// TwinCAT 3 PLC project Command_Pattern
// ProgramVersion: 3.1.4024.0
// libraries:
//   Tc2_Standard, * (Beckhoff Automation GmbH)
//   Tc2_System, * (Beckhoff Automation GmbH)
//   Tc2_Utilities, * (Beckhoff Automation GmbH)
//   Tc3_Module, * (Beckhoff Automation GmbH)
// project tree:
//   Commands/ AxisDisableCommand.TcPOU, AxisEnableCommand.TcPOU, AxisMoveCommand.TcPOU, ITF_Command.TcIO
//   Invoker/ Invoker.TcPOU
//   / PlcTask.TcTTO
//   POUs/ MAIN.TcPOU
//   Reciever/ FB_Axis.TcPOU, ITF_Axis.TcIO
// (motion and I/O tree: see PLC project simple_factory_pattern)
// real-time tasks:
//   TASK PlcTask: cycle T#10ms, priority 20, ADS port 350
//   TASK PlcTask1: cycle T#10ms, priority 21, ADS port 351
//   TASK PlcTask2: cycle T#10ms, priority 22, ADS port 352
//   TASK PlcTask3: cycle T#10ms, priority 23, ADS port 353
//   TASK PlcTask4: cycle T#10ms, priority 24, ADS port 354
//   TASK PlcTask5: cycle T#10ms, priority 25, ADS port 355
//   TASK PlcTask6: cycle T#10ms, priority 26, ADS port 356
//   TASK PlcTask7: cycle T#10ms, priority 27, ADS port 357
//   TASK PlcTask8: cycle T#10ms, priority 28, ADS port 358
//   TASK PlcTask9: cycle T#10ms, priority 29, ADS port 359
//   TASK PlcTask10: cycle T#10ms, priority 30, ADS port 360
//   TASK PlcTask11: cycle T#10ms, priority 31, ADS port 361

CONFIGURATION Command_Pattern
    RESOURCE PLC ON TwinCAT3
        TASK PlcTask(INTERVAL := T#10ms, PRIORITY := 30);
        PROGRAM MAIN WITH PlcTask : MAIN;
    END_RESOURCE
END_CONFIGURATION

// ---- Commands/ITF_Command.TcIO
INTERFACE ITF_Command

METHOD Execute : BOOL
VAR_INPUT
END_VAR
END_METHOD

END_INTERFACE

// ---- Reciever/ITF_Axis.TcIO
INTERFACE ITF_Axis

METHOD Disable : BOOL
VAR_INPUT
END_VAR
END_METHOD

METHOD Enable : BOOL
VAR_INPUT
	EnablePositive : BOOL;
	EnableNegative : BOOL;
	Override : LREAL;
END_VAR
END_METHOD

METHOD MoveToPosition : BOOL
VAR_INPUT
	Position : LREAL;
	Velocity : LREAL;
END_VAR
END_METHOD

END_INTERFACE

// ---- POUs/MAIN.TcPOU
PROGRAM MAIN
VAR
	Axis1 : FB_Axis;
	DisableCmd : AxisDisableCommand := (MyAxis := Axis1);
	EnableCmd : AxisEnableCommand := (MyAxis := Axis1);
	MoveCmd : AxisMoveCommand := (MyAxis := Axis1);
	EnableButton : Invoker;
	DisableButton : Invoker;
	MoveButton : Invoker;
	Initialised: BOOL;
	Enable: BOOL;
	Disable: BOOL;
	MoveAxis: BOOL;
END_VAR

IF NOT Initialised THEN
	EnableButton.SetCommand(MyCommand := EnableCmd);
	DisableButton.SetCommand(MyCommand := DisableCmd);
	MoveButton.SetCommand(MyCommand := MoveCmd);
	Initialised := TRUE;
END_IF

IF Enable THEN
	IF EnableButton.ExecuteCommand() THEN
		Enable := FALSE;
	END_IF
END_IF

IF Disable THEN
	IF DisableButton.ExecuteCommand() THEN
		Disable := FALSE;
	END_IF
END_IF

IF MoveAxis THEN
	IF MoveButton.ExecuteCommand() THEN
		MoveAxis := FALSE;
	END_IF
END_IF

END_PROGRAM

// ---- Reciever/FB_Axis.TcPOU
FUNCTION_BLOCK PUBLIC FB_Axis IMPLEMENTS ITF_Axis
VAR
	testString : STRING;
END_VAR

METHOD Disable : BOOL
VAR_INPUT
END_VAR
ADSLOGSTR( msgCtrlMask := ADSLOG_MSGTYPE_ERROR OR ADSLOG_MSGTYPE_MSGBOX,
			msgFmtStr :='Axis Disabling',
 			strArg := '');
END_METHOD

METHOD Enable : BOOL
VAR_INPUT
	EnablePositive : BOOL;
	EnableNegative : BOOL;
	Override : LREAL;
END_VAR
testString := '';
testString := CONCAT(testString, '[');
testString := CONCAT(testString, BOOL_TO_STRING(EnablePositive));
testString := CONCAT(testString, ']');
testString := CONCAT(testString, '[');
testString := CONCAT(testString, BOOL_TO_STRING(EnableNegative));
testString := CONCAT(testString, ']');
testString := CONCAT(testString, '[');
testString := CONCAT(testString, LREAL_TO_STRING(Override));
testString := CONCAT(testString, ']');

ADSLOGSTR( msgCtrlMask := ADSLOG_MSGTYPE_ERROR OR ADSLOG_MSGTYPE_MSGBOX,
			msgFmtStr :='Axis Enabling: %s',
 			strArg := testString);
END_METHOD

METHOD MoveToPosition : BOOL
VAR_INPUT
	Position : LREAL;
	Velocity : LREAL;
END_VAR
testString := '';
testString := CONCAT(testString, '[');
testString := CONCAT(testString, LREAL_TO_STRING(Position));
testString := CONCAT(testString, ']');
testString := CONCAT(testString, '[');
testString := CONCAT(testString, LREAL_TO_STRING(Velocity));
testString := CONCAT(testString, ']');

ADSLOGSTR( msgCtrlMask := ADSLOG_MSGTYPE_ERROR OR ADSLOG_MSGTYPE_MSGBOX,
			msgFmtStr :='Axis Moving: %s',
 			strArg := testString);
END_METHOD

END_FUNCTION_BLOCK

// ---- Commands/AxisDisableCommand.TcPOU
FUNCTION_BLOCK AxisDisableCommand IMPLEMENTS ITF_Command
VAR
	_reciever : ITF_Axis;
END_VAR

METHOD Execute : BOOL
IF _reciever <> 0 THEN
	_reciever.Disable();
END_IF
END_METHOD

PROPERTY MyAxis : ITF_Axis
GET
MyAxis := _reciever;
END_GET
SET
_reciever := MyAxis;
END_SET
END_PROPERTY

END_FUNCTION_BLOCK

// ---- Commands/AxisEnableCommand.TcPOU
FUNCTION_BLOCK AxisEnableCommand IMPLEMENTS ITF_Command
VAR
	_reciever : ITF_Axis;
	_enablePositive : BOOL;
	_enableNegative : BOOL;
	_override : LREAL;
END_VAR

PROPERTY EnableNegative : BOOL
GET
EnableNegative := _enableNegative;
END_GET
SET
_enableNegative := EnableNegative;
END_SET
END_PROPERTY

PROPERTY EnablePositive : BOOL
GET
EnablePositive := _enablePositive;
END_GET
SET
_enablePositive := EnablePositive;
END_SET
END_PROPERTY

METHOD Execute : BOOL
IF _reciever <> 0 THEN
	_reciever.Enable(_enablePositive, _enableNegative, _override);
END_IF
END_METHOD

PROPERTY MyAxis : ITF_Axis
GET
MyAxis := _reciever;
END_GET
SET
_reciever := MyAxis;
END_SET
END_PROPERTY

PROPERTY Override : LREAL
GET
Override := _override;
END_GET
SET
_override := Override;
END_SET
END_PROPERTY

END_FUNCTION_BLOCK

// ---- Commands/AxisMoveCommand.TcPOU
FUNCTION_BLOCK AxisMoveCommand IMPLEMENTS ITF_Command
VAR
	_reciever : ITF_Axis;
	_position : LREAL;
	_velocity : LREAL;
END_VAR

METHOD Execute : BOOL
IF _reciever <> 0 THEN
	_reciever.MoveToPosition(Position := _position, Velocity := _velocity);
END_IF
END_METHOD

PROPERTY MyAxis : ITF_Axis
GET
MyAxis := _reciever;
END_GET
SET
_reciever := MyAxis;
END_SET
END_PROPERTY

PROPERTY Position : LREAL
GET
Position := _position;
END_GET
SET
_position := Position;
END_SET
END_PROPERTY

PROPERTY Velocity : LREAL
GET
Velocity := _velocity;
END_GET
SET
_velocity := Velocity;
END_SET
END_PROPERTY

END_FUNCTION_BLOCK

// ---- Invoker/Invoker.TcPOU
FUNCTION_BLOCK Invoker
VAR
	_myCommand : ITF_Command;
END_VAR

METHOD ExecuteCommand : BOOL
VAR_INPUT
END_VAR
_myCommand.Execute();
ExecuteCommand := true;
END_METHOD

METHOD SetCommand : BOOL
VAR_INPUT
	MyCommand : ITF_Command;
END_VAR
_myCommand := MyCommand;
SetCommand := true;
END_METHOD

END_FUNCTION_BLOCK
